// TIA Portal project "Project4" (V16)

(* hardware
DEVICE "S7300/ET200M station_1"  S7-300 station
   slot 0: "Rail_0"  Rail  6ES7 390-1***0-0AA0
   slot 2: "PLC_1"  CPU 315-2 PN/DP  6ES7 315-2EH14-0AB0  V3.2
      slot 2: "PROFINET interface_1"  PN-IO
         slot 1: "Port_1"  Port
         slot 2: "Port_2"  Port
*)

// ===== PLC "PLC_1"  CPU 315-2 PN/DP =====

VAR_GLOBAL   // PLC tag table "Default tag table"
   "Tag_1" AT %I0.1 : Bool;
   "Tag_2" AT %I1.1 : Bool;
   "Tag_3" AT %T1 : Timer;
   "Tag_4" AT %MW10 : Word;
   "Tag_5" AT %MW20 : Word;
   "Tag_6" AT %Q0.1 : Bool;
   "Tag_7" AT %I0.2 : Bool;
   "Tag_8" AT %I1.2 : Bool;
   "Tag_9" AT %T2 : Timer;
   "Tag_10" AT %MW12 : Word;
   "Tag_11" AT %MW22 : Word;
   "Tag_12" AT %Q0.2 : Bool;
   "Tag_13" AT %I0.3 : Bool;
   "Tag_14" AT %I1.3 : Bool;
   "Tag_15" AT %T3 : Timer;
   "Tag_16" AT %MW14 : Word;
   "Tag_17" AT %MW24 : Word;
   "Tag_18" AT %Q0.3 : Bool;
   "Tag_19" AT %I0.4 : Bool;
   "Tag_20" AT %T4 : Timer;
   "Tag_21" AT %MW16 : Word;
   "Tag_22" AT %MW26 : Word;
   "Tag_23" AT %Q0.4 : Bool;
   "Tag_24" AT %I1.4 : Bool;
   "Tag_25" AT %I0.5 : Bool;
   "Tag_26" AT %I1.5 : Bool;
   "Tag_27" AT %T5 : Timer;
   "Tag_28" AT %MW18 : Word;
   "Tag_29" AT %MW28 : Word;
   "Tag_30" AT %I0.6 : Bool;
   "Tag_31" AT %T7 : Timer;
   "Tag_32" AT %T6 : Timer;
   "Tag_33" AT %Q0.6 : Bool;
   "Tag_34" AT %Q0.7 : Bool;
   "Tag_35" AT %Q0.5 : Bool;
   "Tag_36" AT %I0.7 : Bool;
   "Tag_37" AT %M0.0 : Bool;
   "Tag_38" AT %T8 : Timer;
   "Tag_39" AT %C1 : Counter;
   "Tag_40" AT %MW30 : Word;
   "Tag_41" AT %Q1.0 : Bool;
   "Tag_42" AT %Q1.1 : Bool;
   "Tag_43" AT %Q1.2 : Bool;
END_VAR

ORGANIZATION_BLOCK "Main"   // OB1, LAD
TITLE = "Main Program Sweep (Cycle)"
{ S7_Optimized_Access := 'FALSE' }
VERSION : 0.1
   VAR_TEMP
      OB1_EV_CLASS : Byte;   // Bits 0-3 = 1 (Coming event), Bits 4-7 = 1 (Event class 1)
      OB1_SCAN_1 : Byte;   // 1 (Cold restart scan 1 of OB 1), 3 (Scan 2-n of OB 1)
      OB1_PRIORITY : Byte;   // Priority of OB Execution
      OB1_OB_NUMBR : Byte;   // 1 (Organization block 1, OB1)
      OB1_RESERVED_1 : Byte;   // Reserved for system
      OB1_RESERVED_2 : Byte;   // Reserved for system
      OB1_PREV_CYCLE : Int;   // Cycle time of previous OB1 scan (milliseconds)
      OB1_MIN_CYCLE : Int;   // Minimum cycle time of OB1 (milliseconds)
      OB1_MAX_CYCLE : Int;   // Maximum cycle time of OB1 (milliseconds)
      OB1_DATE_TIME : Date_And_Time;   // Date and time OB1 started
   END_VAR
   VAR_TEMP   // added for the SCL form of the ladder/FBD networks
      _w1 : Bool;
      _s5time1 : S5Time;
   END_VAR
BEGIN

REGION Network 1: Pulse Timer (SP)
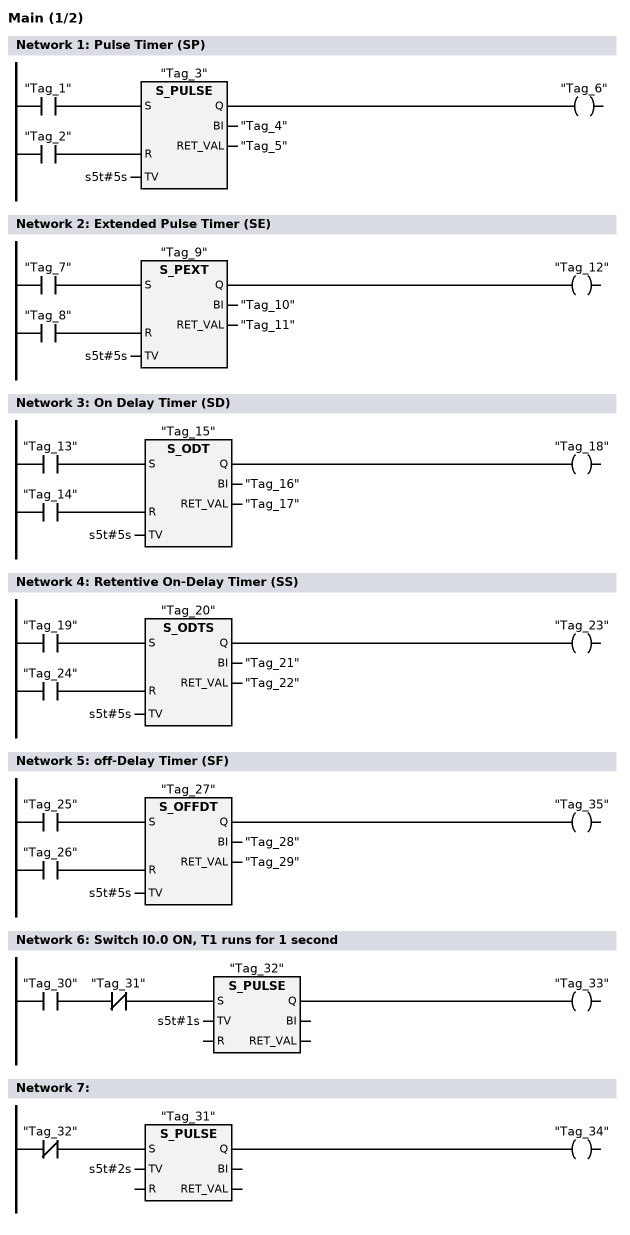
   RUNG wire#powerrail
      Contact( "Tag_1" )
      S_PULSE(T_NO := "Tag_3", R := wire#w1, TV := s5t#5s, BI => "Tag_4", RET_VAL => "Tag_5")
      Coil( "Tag_6" )
   END_RUNG
   RUNG wire#powerrail
      Contact( "Tag_2" )
   END_RUNG wire#w1
   // the same network as SCL:
   "Tag_5" := S_PULSE(T_NO := "Tag_3", S := "Tag_1", R := "Tag_2", TV := s5t#5s, Q => #_w1, BI => "Tag_4");
   "Tag_6" := #_w1;
END_REGION

REGION Network 2: Extended Pulse Timer (SE)
   RUNG wire#powerrail
      Contact( "Tag_7" )
      S_PEXT(T_NO := "Tag_9", R := wire#w1, TV := s5t#5s, BI => "Tag_10", RET_VAL => "Tag_11")
      Coil( "Tag_12" )
   END_RUNG
   RUNG wire#powerrail
      Contact( "Tag_8" )
   END_RUNG wire#w1
   // the same network as SCL:
   "Tag_11" := S_PEXT(T_NO := "Tag_9", S := "Tag_7", R := "Tag_8", TV := s5t#5s, Q => #_w1, BI => "Tag_10");
   "Tag_12" := #_w1;
END_REGION

REGION Network 3: On Delay Timer (SD)
   RUNG wire#powerrail
      Contact( "Tag_13" )
      S_ODT(T_NO := "Tag_15", R := wire#w1, TV := s5t#5s, BI => "Tag_16", RET_VAL => "Tag_17")
      Coil( "Tag_18" )
   END_RUNG
   RUNG wire#powerrail
      Contact( "Tag_14" )
   END_RUNG wire#w1
   // the same network as SCL:
   "Tag_17" := S_ODT(T_NO := "Tag_15", S := "Tag_13", R := "Tag_14", TV := s5t#5s, Q => #_w1, BI => "Tag_16");
   "Tag_18" := #_w1;
END_REGION

REGION Network 4: Retentive On-Delay Timer (SS)
   RUNG wire#powerrail
      Contact( "Tag_19" )
      S_ODTS(T_NO := "Tag_20", R := wire#w1, TV := s5t#5s, BI => "Tag_21", RET_VAL => "Tag_22")
      Coil( "Tag_23" )
   END_RUNG
   RUNG wire#powerrail
      Contact( "Tag_24" )
   END_RUNG wire#w1
   // the same network as SCL:
   "Tag_22" := S_ODTS(T_NO := "Tag_20", S := "Tag_19", R := "Tag_24", TV := s5t#5s, Q => #_w1, BI => "Tag_21");
   "Tag_23" := #_w1;
END_REGION

REGION Network 5: off-Delay Timer (SF)
   RUNG wire#powerrail
      Contact( "Tag_25" )
      S_OFFDT(T_NO := "Tag_27", R := wire#w1, TV := s5t#5s, BI => "Tag_28", RET_VAL => "Tag_29")
      Coil( "Tag_35" )
   END_RUNG
   RUNG wire#powerrail
      Contact( "Tag_26" )
   END_RUNG wire#w1
   // the same network as SCL:
   "Tag_29" := S_OFFDT(T_NO := "Tag_27", S := "Tag_25", R := "Tag_26", TV := s5t#5s, Q => #_w1, BI => "Tag_28");
   "Tag_35" := #_w1;
END_REGION

REGION Network 6: Switch I0.0 ON, T1 runs for 1 second
   RUNG wire#powerrail
      Contact( "Tag_30" )
      I_Contact( "Tag_31" )
      S_PULSE(T_NO := "Tag_32", TV := s5t#1s, R :=, BI =>, RET_VAL =>)
      Coil( "Tag_33" )
   END_RUNG
   // the same network as SCL:
   #_s5time1 := S_PULSE(T_NO := "Tag_32", S := "Tag_30" AND NOT "Tag_31", TV := s5t#1s, Q => #_w1);
   "Tag_33" := #_w1;
END_REGION

REGION Network 7
   RUNG wire#powerrail
      I_Contact( "Tag_32" )
      S_PULSE(T_NO := "Tag_31", TV := s5t#2s, R :=, BI =>, RET_VAL =>)
      Coil( "Tag_34" )
   END_RUNG
   // the same network as SCL:
   #_s5time1 := S_PULSE(T_NO := "Tag_31", S := NOT "Tag_32", TV := s5t#2s, Q => #_w1);
   "Tag_34" := #_w1;
END_REGION

REGION Network 8: One-cycle pulse generator with On-delay timer
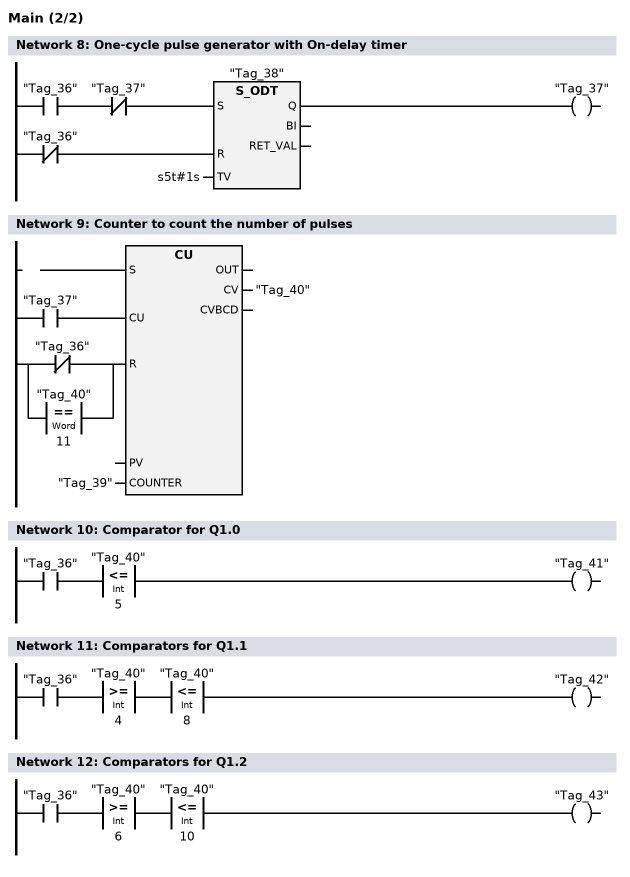
   RUNG wire#powerrail
      Contact( "Tag_36" )
      I_Contact( "Tag_37" )
      S_ODT(T_NO := "Tag_38", R := wire#w1, TV := s5t#1s, BI =>, RET_VAL =>)
      Coil( "Tag_37" )
   END_RUNG
   RUNG wire#powerrail
      I_Contact( "Tag_36" )
   END_RUNG wire#w1
   // the same network as SCL:
   #_s5time1 := S_ODT(T_NO := "Tag_38",
                      S := "Tag_36" AND NOT "Tag_37",
                      R := NOT "Tag_36",
                      TV := s5t#1s,
                      Q => #_w1);
   "Tag_37" := #_w1;
END_REGION

REGION Network 9: Counter to count the number of pulses
   // no SCL statement known for Cu: written as a call
   Cu(cu := "Tag_37", r := NOT "Tag_36" OR ("Tag_40" = 11), "counter" := "Tag_39", cv => "Tag_40");
END_REGION

REGION Network 10: Comparator for Q1.0
   RUNG wire#powerrail
      Contact( "Tag_36" )
      { S7_Templates := "SrcType := Int" } LE_Contact(in1 := "Tag_40", in2 := 5)
      Coil( "Tag_41" )
   END_RUNG
   // the same network as SCL:
   "Tag_41" := "Tag_36" AND ("Tag_40" <= 5);
END_REGION

REGION Network 11: Comparators for Q1.1
   RUNG wire#powerrail
      Contact( "Tag_36" )
      { S7_Templates := "SrcType := Int" } GE_Contact(in1 := "Tag_40", in2 := 4)
      { S7_Templates := "SrcType := Int" } LE_Contact(in1 := "Tag_40", in2 := 8)
      Coil( "Tag_42" )
   END_RUNG
   // the same network as SCL:
   "Tag_42" := "Tag_36" AND ("Tag_40" >= 4) AND ("Tag_40" <= 8);
END_REGION

REGION Network 12: Comparators for Q1.2
   RUNG wire#powerrail
      Contact( "Tag_36" )
      { S7_Templates := "SrcType := Int" } GE_Contact(in1 := "Tag_40", in2 := 6)
      { S7_Templates := "SrcType := Int" } LE_Contact(in1 := "Tag_40", in2 := 10)
      Coil( "Tag_43" )
   END_RUNG
   // the same network as SCL:
   "Tag_43" := "Tag_36" AND ("Tag_40" >= 6) AND ("Tag_40" <= 10);
END_REGION
END_ORGANIZATION_BLOCK